// TwinCAT 3 PLC project RobotsNew
// ProgramVersion: 3.1.4023.0
// libraries:
//   Tc2_Standard, * (Beckhoff Automation GmbH)
//   Tc2_System, * (Beckhoff Automation GmbH)
//   Tc2_Utilities, * (Beckhoff Automation GmbH)
//   Tc3_Module, * (Beckhoff Automation GmbH)
// project tree:
//   DUTs/Robot Tasks/ TaskA21.TcDUT, TaskA22.TcDUT, TaskA26.TcDUT
//   DUTs/Robots/ I_Area2Robot.TcIO, KukaRobot.TcPOU, RobotA21.TcPOU, RobotA22.TcPOU, RobotA26.TcPOU
//   DUTs/ SectionEnum.TcDUT, Watchdog.TcPOU
//   / PlcTask2.TcTTO
//   POUs/ MAIN.TcPOU
// (motion and I/O tree: see PLC project conveyorslinking)
// real-time tasks:
//   TASK PlcTask: cycle T#10ms, priority 20, ADS port 350
//   TASK PlcTask1: cycle T#10ms, priority 21, ADS port 351
//   TASK PlcTask2: cycle T#10ms, priority 22, ADS port 352
//   TASK PlcTask3: cycle T#10ms, priority 23, ADS port 353

CONFIGURATION RobotsNew
    RESOURCE PLC ON TwinCAT3
        TASK PlcTask2(INTERVAL := T#10ms, PRIORITY := 22);
        PROGRAM MAIN WITH PlcTask2 : MAIN;
    END_RESOURCE
END_CONFIGURATION

// ---- DUTs/Robot Tasks/TaskA21.TcDUT
{attribute 'qualified_only'}
//{attribute 'strict'}
{attribute 'to_string'}
TYPE TaskA21 :
(
	IDLE,
	STAGE_BUNK,
	REMOVE_BUNK_FROM_STAGE,
	
	LOAD_BUNK_TOP := 4,
	LOAD_BUNK_SIDE,
	LOAD_BUNK_BOTTOM,
	REMOVE_BUNK_TOP,
	REMOVE_BUNK_SIDE,
	REMOVE_BUNK_BOTTOM,
	
	//GET_CHIPBOARD_FROM_SKID := 11,
	//OFFLOAD_CHIPBOARD,
	PLACE_CHIPBOARD_TOP := 13,
	PLACE_CHIPBOARD_BOTTOM,
	REMOVE_CHIPBOARD_TOP,
	REMOVE_CHIPBOARD_BOTTOM,
	
	FIX_CHIPBOARD_ORIENTATION := 19,
	
	//testing only
	MOVE_HOME := 21,
	MOVE_POSITION1,
	MOVE_POSITION2,
	MOVE_UP,
	MOVE_DOWN,
	
	DIRECT_BUNK_TOP := 27,
	DIRECT_BUNK_SIDE,
	DIRECT_BUNK_BOTTOM,
	
	INSPECT_BUNK := 31,
	INSPECT_CHIPBOARD,
	
	TOOL_CHANGE_BUNK := 34,
	TOOL_CHANGE_CHIPBOARD,
	
	size
);
END_TYPE

// ---- DUTs/Robot Tasks/TaskA22.TcDUT
{attribute 'qualified_only'}
{attribute 'to_string'}
//{attribute 'strict'}
TYPE TaskA22 :
(
	IDLE,
	
	LOAD_CARDBOARD_TOP, //flat cardboards
	LOAD_CARDBOARD_BOTTOM,
	LOAD_CARDBOARD_SIDE,
	REMOVE_CARDBOARD_TOP,
	REMOVE_CARDBOARD_BOTTOM,
	REMOVE_CARDBOARD_SIDE,
	
	TRANSFER_TO_BENDER := 9, //corner cardboards
	TRANSFER_TO_OVERHEAD,
	REMOVE_CARDBOARD_FROM_BENDER,
	LOAD_BENDER_TO_UPPER_CORNER,
	LOAD_BENDER_TO_LOWER_CORNER,
	LOAD_OVERHEAD_TO_UPPER_CORNER,
	LOAD_OVERHEAD_TO_LOWER_CORNER,
	
	REMOVE_CARDBOARD_UPPER_CORNER,
	REMOVE_CARDBOARD_LOWER_CORNER,
	REMOVE_CARDBOARD_OVERHEAD := 18,
	
	LOAD_CORNER_GUARD_UPPER := 20, //corner guards
	LOAD_CORNER_GUARD_LOWER,
	REMOVE_CORNER_GUARD_UPPER,
	REMOVE_CORNER_GUARD_LOWER,
	
	size
);
END_TYPE

// ---- DUTs/Robot Tasks/TaskA26.TcDUT
{attribute 'qualified_only'}
{attribute 'to_string'}
//{attribute 'strict'}
TYPE TaskA26 :
(
	IDLE,
	PICK_SPACER,
	
	size
);
END_TYPE

// ---- DUTs/SectionEnum.TcDUT
{attribute 'qualified_only'}
TYPE SectionEnum :
(
	NULL_SECTION := -1,
	PAPER,
	CARDBOARD_CORNERGUARD,
	CHIPBOARD,
	WOOD_BUNK,
	OUTPUT,
	
	size
);
END_TYPE

// ---- DUTs/Robots/I_Area2Robot.TcIO
INTERFACE I_Area2Robot

//{attribute 'monitoring' := 'variable'}
{attribute 'monitoring' := 'call'}
PROPERTY Busy : BOOL
GET
END_GET
END_PROPERTY

METHOD clearCommand : BOOL
VAR_INPUT
END_VAR
END_METHOD

//{attribute 'monitoring' := 'variable'}
{attribute 'monitoring' := 'call'}
PROPERTY Done : BOOL
GET
END_GET
END_PROPERTY

{attribute 'monitoring' := 'call'}
PROPERTY Ready : BOOL
GET
END_GET
END_PROPERTY

METHOD release : BOOL
VAR_INPUT
	sectionReservation : SectionEnum;
END_VAR
END_METHOD

METHOD reserve : BOOL
VAR_INPUT
	reserveRequest : SectionEnum;
END_VAR
(*
this method exists because chipboard and wood bunk operations use the same robot
both sections need to check if the robot is open to commands before use
*)
END_METHOD

{attribute 'monitoring' := 'call'}
PROPERTY Reserved : BOOL
GET
END_GET
END_PROPERTY

METHOD reset : BOOL
END_METHOD

METHOD stop : BOOL
VAR_INPUT
END_VAR
END_METHOD

END_INTERFACE

// ---- POUs/MAIN.TcPOU
PROGRAM MAIN
VAR_OUTPUT
	localTime : TIMESTRUCT;
END_VAR
VAR
	r21 : RobotA21;
	r22 : RobotA22;
	r26 : RobotA26;
END_VAR

END_PROGRAM

// ---- DUTs/Robots/RobotA21.TcPOU
FUNCTION_BLOCK RobotA21 EXTENDS KukaRobot
VAR_INPUT
	strapSafety : BOOL;
END_VAR
VAR_OUTPUT //from outputs array
	taskID AT %Q* : TaskA21;
	param1 AT %Q* : INT;
	param2 AT %Q* : INT;
	Xmm AT %Q* : INT;
	Ymm AT %Q* : INT;
	Zmm AT %Q* : INT;
	angle AT %Q* : INT;
	stagingOccupancy AT %Q* : INT;
	insertionSuctionStatus : INT;
	magazineStatus AT %Q* : INT; //unused
	inspectionValue AT %Q* : INT;
	
	strapSafetyOut : BOOL;
END_VAR
VAR_OUTPUT //from inputs array
	tool : SectionEnum := SectionEnum.WOOD_BUNK;
	suspendedMaterial : STRING;
	
	completedTask AT %I* : TaskA21;
	eoatDistance AT %I* : INT;
	woodBunkAvailability AT %I* : INT;
	chipboardAvailability AT %I* : INT;
	materialAtHoldingPosition AT %I* : INT;
	
	strapSafetyIn AT %I* : BOOL;
END_VAR
VAR
	reservationEnum : SectionEnum;
	hmiTask : STRING;
	hmiTool : STRING;
END_VAR
(*
extends KukaRobot
	assigns descriptive labels to each IO group from the array
	additional section-specific methods to get/set IO groups
*)

{warning disable C0195}

SUPER^();

//set the strings to display on the HMI
reservationEnum := reservation;
IF reservationEnum = SectionEnum.NULL_SECTION THEN
	hmiReservation := 'N/A';
ELSE
	hmiReservation := TO_STRING(reservationEnum);
END_IF

hmiTask := TO_STRING(taskID);
hmiTool := TO_STRING(tool);

{attribute 'monitoring' := 'call'}
PROPERTY Busy : BOOL
GET
VAR
	//emptyOutput : ARRAY[1..50] OF INT;
END_VAR
//Busy stays TRUE until outputs are cleared AND completed task has elapsed
//Ready is always inverse of Busy
Busy := taskID <> 0 OR completedTask <> 0;
END_GET
END_PROPERTY

METHOD changeEOAT : BOOL
VAR_INPUT
	targetTool : SectionEnum;
END_VAR
IF tool = targetTool THEN
	changeEOAT := TRUE;
	
ELSE
	
	CASE targetTool OF
		SectionEnum.CHIPBOARD:	taskID := TaskA21.TOOL_CHANGE_CHIPBOARD;
		SectionEnum.WOOD_BUNK:	taskID := TaskA21.TOOL_CHANGE_BUNK;
	END_CASE
	
END_IF
END_METHOD

METHOD clearCommand : BOOL
VAR_INPUT
END_VAR
taskID := 0;
param1 := 0;
param2 := 0;
Xmm := 0;
Ymm := 0;
Zmm := 0;;
angle := 0;
stagingOccupancy := 0;
insertionSuctionStatus := 0;
magazineStatus := 0;
inspectionValue := 0;
END_METHOD

{attribute 'monitoring' := 'call'}
PROPERTY Done : BOOL
GET
Done :=
	completedTask = taskID AND
	taskID <> 0 AND
	completedTask <> 0;
END_GET
END_PROPERTY

{attribute 'monitoring' := 'call'}
PROPERTY HoldMaterial : STRING
GET
HoldMaterial := suspendedMaterial;
END_GET
SET
suspendedMaterial := HoldMaterial;
END_SET
END_PROPERTY

{attribute 'monitoring' := 'call'}
PROPERTY Ready : BOOL
GET
Ready := taskID = 0 AND completedTask = 0;
END_GET
END_PROPERTY

METHOD setParameters : BOOL
VAR_INPUT
	newTaskID : INT;
	newParam1 : INT;
	newParam2 : INT;
	newXmm : INT;
	newYmm : INT;
	newZmm : INT;
	newAngle : INT;
	newStagingOccupancy : INT;
	newInsertionSuctionStatus : INT;
	newMagazineStatus : INT; //unused
	newInspectionValue : INT;
END_VAR
VAR_INPUT
	newStrapSafety : BOOL;
END_VAR
taskID := newTaskID;
param1 := newParam1;
param2 := newParam2;
Xmm := newXmm;
Ymm := newYmm;
Zmm := newZmm;
angle := newAngle;

stagingOccupancy := newStagingOccupancy;
stagingOccupancy.15 := newStrapSafety;

insertionSuctionStatus := newInsertionSuctionStatus;
magazineStatus := newMagazineStatus;
inspectionValue := newInspectionValue;
END_METHOD

END_FUNCTION_BLOCK

// ---- DUTs/Robots/KukaRobot.TcPOU
FUNCTION_BLOCK ABSTRACT KukaRobot
VAR_INPUT
	bEnable : BOOL; //enables the robot
	abort : BOOL; //disables the robot
END_VAR
VAR_OUTPUT
	(*
	forceStop AT %Q* : BOOL;
	resetSignal AT %Q* : BOOL;
	*)
	
	reservation : INT := 0;
	
	error : BOOL;
	errorID : DINT;
END_VAR
VAR
	heartbeat : Watchdog;
	
	disconnected AT %I* : BOOL;
	toggleBit AT %I* : BOOL;
	
	hmiReservation : STRING;
END_VAR
(*
generic KUKA robot with 20 WORD outputs and 20 WORD inputs, connected to Beckhoff IPC via EL6692 or EL6695 EtherCAT bridge
includes minimal diagnostics to detect if robot is offline
robots should always be reserved before sending a task
*)

heartbeat(
	enable:= NOT disconnected,
	toggleBit:= toggleBit,
	timeoutWidth:= T#200MS,
	timeout=> );

error := //add any addition conditions with OR
	disconnected OR
	heartbeat.timeout;
	
//bEnable must be TRUE and abort must be FALSE for the robot to function
IF (*NOT bEnable OR*) abort THEN //bEnable is not used for now, but abort is
	stop();
END_IF

//{attribute 'monitoring' := 'variable'}
{attribute 'monitoring' := 'call'}
PROPERTY ABSTRACT Busy : BOOL
GET
END_GET
END_PROPERTY

METHOD ABSTRACT clearCommand : BOOL
VAR_INPUT
END_VAR
END_METHOD

//{attribute 'monitoring' := 'variable'}
{attribute 'monitoring' := 'call'}
PROPERTY ABSTRACT Done : BOOL
GET
END_GET
END_PROPERTY

{attribute 'monitoring' := 'call'}
PROPERTY ABSTRACT Ready : BOOL
GET
END_GET
END_PROPERTY

METHOD release : BOOL
VAR_INPUT
	sectionReservation : INT;
END_VAR
IF reservation = sectionReservation THEN
	reservation := 0;
	release := TRUE;
END_IF
END_METHOD

METHOD reserve : BOOL
VAR_INPUT
	reserveRequest : INT;
END_VAR
(*
this method exists because chipboard and wood bunk operations use the same robot
both sections need to check if the robot is open to commands before use
*)
IF Reserved AND reservation = reserveRequest THEN
	reserve := TRUE;

ELSIF NOT Reserved THEN
	reservation := reserveRequest;
	reserve := TRUE;

END_IF
END_METHOD

{attribute 'monitoring' := 'call'}
PROPERTY Reserved : BOOL
GET
Reserved := reservation <> 0;
END_GET
END_PROPERTY

METHOD reset : BOOL
abort := TRUE;
clearCommand();
END_METHOD

METHOD resume : BOOL
VAR_INPUT
END_VAR
//forceStop := FALSE;
IF NOT error AND errorID = 0 THEN
	resume := TRUE;
	abort := FALSE;
END_IF
END_METHOD

METHOD stop : BOOL
VAR_INPUT
END_VAR
//forceStop := TRUE;
abort := TRUE;
clearCommand();

stop := TRUE;
END_METHOD

END_FUNCTION_BLOCK

// ---- DUTs/Watchdog.TcPOU
FUNCTION_BLOCK Watchdog
VAR_INPUT
	enable : BOOL := TRUE; //watchdog can be disabled if needed
	
	toggleBit : BOOL;
	timeoutWidth : TIME := T#3S;
END_VAR
VAR_OUTPUT
	timeout : BOOL;
	prevMsgTimestamp : TIMESTRUCT;
END_VAR
VAR	
	timer : TON;
	memoryBit : BOOL;
END_VAR

timer(
	IN:= enable AND (memoryBit = toggleBit), 
	PT:= timeoutWidth, 
	Q=> timeout, 
	ET=> );
	
IF enable AND memoryBit <> toggleBit THEN
	prevMsgTimestamp := MAIN.localTime;
END_IF

memoryBit := toggleBit;

END_FUNCTION_BLOCK

// ---- DUTs/Robots/RobotA22.TcPOU
FUNCTION_BLOCK RobotA22 EXTENDS KukaRobot
VAR_INPUT
	wrapSafety AT %Q* : BOOL;
END_VAR
VAR_OUTPUT //from outputs array
	taskID AT %Q* : TaskA22;
	param1 AT %Q* : INT;
	param2 AT %Q* : INT;
	Xmm AT %Q* : INT;
	Ymm AT %Q* : INT;
	Zmm AT %Q* : INT;
	angle AT %Q* : INT;
	foldPosition0 AT %Q* : INT;
	foldPosition1 AT %Q* : INT;
END_VAR
VAR_OUTPUT //from inputs array
	tool : SectionEnum := SectionEnum.CARDBOARD_CORNERGUARD;
	suspendedMaterial : STRING;
	
	completedTask AT %I* : TaskA22;
	eoatDistance AT %I* : INT;
	cardboardAvailability AT %I* : INT;
	cornerGuardAvailability AT %I* : INT;
	materialAtHoldingPosition AT %I* : INT;
	//grp6	
	wrapSafetyIn AT %I* : BOOL;
END_VAR
VAR //HMI data
	reservationEnum : SectionEnum;
	hmiTask : STRING;
	hmiTool : STRING;
END_VAR

{warning disable C0195}

SUPER^();

reservationEnum := reservation;
IF reservationEnum = SectionEnum.NULL_SECTION THEN
	hmiReservation := 'N/A';
ELSE
	hmiReservation := TO_STRING(reservationEnum);
END_IF

hmiTask := TO_STRING(taskID);
hmiTool := TO_STRING(tool);

{attribute 'monitoring' := 'call'}
PROPERTY Busy : BOOL
GET
VAR
	//emptyOutput : ARRAY[1..50] OF INT;
END_VAR
//Busy stays TRUE until outputs are cleared AND completed task has elapsed
//Ready is always inverse of Busy
Busy := taskID <> 0 OR completedTask <> 0;
END_GET
END_PROPERTY

METHOD changeEOAT : BOOL
VAR_INPUT
	targetTool : SectionEnum;
END_VAR
//fill in IO here

changeEOAT := TRUE;
END_METHOD

METHOD clearCommand : BOOL
VAR_INPUT
END_VAR
taskID := 0;
param1 := 0;
param2 := 0;
Xmm := 0;
Ymm := 0;
Zmm := 0;
angle := 0;
foldPosition0 := 0;
foldPosition1 := 0;
END_METHOD

{attribute 'monitoring' := 'call'}
PROPERTY Done : BOOL
GET
Done :=
	completedTask = taskID AND
	taskID <> 0 AND
	completedTask <> 0;
END_GET
END_PROPERTY

{attribute 'monitoring' := 'call'}
PROPERTY HoldMaterial : STRING
GET
HoldMaterial := suspendedMaterial;
END_GET
SET
suspendedMaterial := HoldMaterial;
END_SET
END_PROPERTY

{attribute 'monitoring' := 'call'}
PROPERTY Ready : BOOL
GET
Ready := taskID = 0 AND completedTask = 0;
END_GET
END_PROPERTY

METHOD setParameters : BOOL
VAR_INPUT
	newTaskID : INT;
	newParam1 : INT;
	newParam2 : INT;
	newXmm : INT;
	newYmm : INT;
	newZmm : INT;
	newAngle : INT;
	newFoldPos0 : INT;
	newFoldPos1 : INT;
END_VAR
VAR_INPUT
	newWrapSafety : BOOL;
END_VAR
taskID := newTaskID;
param1 := newParam1;
param2 := newParam2;
Xmm := newXmm;
Ymm := newYmm;
Zmm := newZmm;
angle := newAngle;
foldPosition0 := newFoldPos0;
foldPosition1 := newFoldPos1;

wrapSafety := newWrapSafety;
END_METHOD

END_FUNCTION_BLOCK

// ---- DUTs/Robots/RobotA26.TcPOU
FUNCTION_BLOCK RobotA26 EXTENDS KukaRobot
VAR_INPUT
	conveyorSafety : BOOL;
END_VAR
VAR_OUTPUT //from outputs array
	{warning disable C0195}
	taskID AT %Q* : TaskA26;
	param1 AT %Q* : INT; //position number (1..6)
	param2 AT %Q* : INT;
	
	strapSafetyOut : BOOL;
END_VAR
VAR_OUTPUT //from inputs array
	tool : SectionEnum := SectionEnum.WOOD_BUNK;
	suspendedMaterial : STRING;
	
	completedTask AT %I* : TaskA26;
	eoatDistance AT %I* : INT;
	
	conveyorSafetyIn : BOOL;
END_VAR
VAR
	reservationEnum : SectionEnum;
	hmiTask : STRING;
	hmiTool : STRING;
END_VAR
(*
extends KukaRobot
	assigns descriptive labels to each IO group from the array
	additional section-specific methods to get/set IO groups
*)

{warning disable C0195}

SUPER^();

reservationEnum := reservation;
IF reservationEnum = SectionEnum.NULL_SECTION THEN
	hmiReservation := 'N/A';
ELSE
	hmiReservation := TO_STRING(reservationEnum);
END_IF

hmiTask := TO_STRING(taskID);
hmiTool := TO_STRING(tool);

{attribute 'monitoring' := 'call'}
PROPERTY Busy : BOOL
GET
VAR
	//emptyOutput : ARRAY[1..50] OF INT;
END_VAR
//Busy stays TRUE until outputs are cleared AND completed task has elapsed
//Ready is always inverse of Busy
Busy := taskID <> 0 OR completedTask <> 0;
END_GET
END_PROPERTY

METHOD clearCommand : BOOL
VAR_INPUT
END_VAR
taskID := 0;
param1 := 0;
param2 := 0;
END_METHOD

{attribute 'monitoring' := 'call'}
PROPERTY Done : BOOL
GET
Done :=
	completedTask = taskID AND
	taskID <> 0 AND
	completedTask <> 0;
END_GET
END_PROPERTY

{attribute 'monitoring' := 'call'}
PROPERTY HoldMaterial : STRING
GET
HoldMaterial := suspendedMaterial;
END_GET
SET
suspendedMaterial := HoldMaterial;
END_SET
END_PROPERTY

{attribute 'monitoring' := 'call'}
PROPERTY Ready : BOOL
GET
Ready := taskID = 0 AND completedTask = 0 AND NOT error;
END_GET
END_PROPERTY

METHOD setParameters : BOOL
VAR_INPUT
	newTaskID : INT;
	newParam1 : INT;
	newParam2 : INT;
END_VAR
VAR_INPUT
	newConveyorSafety : BOOL;
END_VAR
taskID := newTaskID;
param1 := newParam1;
param2 := newParam2;

//missing newConveyorSafety
END_METHOD

END_FUNCTION_BLOCK
